FUNCTION_BLOCK FB_ProfidriveTelegram1_Test EXTENDS TcUnit.FB_TestSuite

Test_ProcessDataControl();
Test_ProcessDataStatus();

METHOD Test_ProcessDataControl : REFERENCE TO FB_Test
VAR
	fbDrive 					: FB_ProfidriveTelegram1;
	
	nExpectedSTW1 				: WORD;
	nExpectedNSOLL				: INT;
	nActualSTW1 				: WORD;
	nActualNSOLL				: INT;	
	
	aExpectedControlData 		: ARRAY[1..4] OF BYTE;
	aExpectedStatusData 		: ARRAY[1..4] OF BYTE;
END_VAR
TEST('Assign Process data Control');

//Arrange
nExpectedSTW1 := 16#A1B2;
nExpectedNSOLL 	:= UINT_TO_INT(16#C3D4);
F_Memcpy(ADR(aExpectedControlData), ADR(nExpectedSTW1), 2, FALSE);
F_Memcpy(ADR(aExpectedControlData) + 2, ADR(nExpectedNSOLL), 2, FALSE);
fbDrive.AssignProcessData(aExpectedControlData, aExpectedStatusData);

//Act
fbDrive.GetControlData();

//Assert
F_Memcpy(ADR(nActualSTW1), ADR(fbDrive.stControl), 2, FALSE);
F_Memcpy(ADR(nActualNSOLL), ADR(fbDrive.stControl) + 2, 2, FALSE);

AssertEquals(Expected := nExpectedSTW1,
             Actual := nActualSTW1,
             Message := 'nSTW1 is not correct');
	 
AssertEquals(Expected := nExpectedNSOLL,
             Actual := nActualNSOLL,
             Message := 'nNSOLL is not correct');	

TEST_FINISHED();


TEST('Assign Process data Control Swap');

//Arrange
nExpectedSTW1 := 16#C3F3;
nExpectedNSOLL 	:= UINT_TO_INT(16#C3F3);
F_Memcpy(ADR(aExpectedControlData), ADR(nExpectedSTW1), 2, TRUE);
F_Memcpy(ADR(aExpectedControlData) + 2, ADR(nExpectedNSOLL), 2, TRUE);

fbDrive.stConfig.bSwapProcessData := TRUE;
fbDrive.AssignProcessData(aExpectedControlData, aExpectedStatusData);

//Act
fbDrive.GetControlData();

//Assert
F_Memcpy(ADR(nActualSTW1), ADR(fbDrive.stControl), 2, FALSE);
F_Memcpy(ADR(nActualNSOLL), ADR(fbDrive.stControl) + 2, 2, FALSE);

AssertEquals(Expected := nExpectedSTW1,
             Actual := nActualSTW1,
             Message := 'nSTW1 is not correct');
	 
AssertEquals(Expected := nExpectedNSOLL,
             Actual := nActualNSOLL,
             Message := 'nNSOLL is not correct');	

TEST_FINISHED();
END_METHOD

METHOD Test_ProcessDataStatus : REFERENCE TO FB_Test
VAR
	fbDrive 					: FB_ProfidriveTelegram1;
	
	nExpectedZSW1 				: WORD;
	nExpectedNIST				: INT;	
	nActualZSW1 				: WORD;
	nActualNIST					: INT;	

	aExpectedControlData 		: ARRAY[1..4] OF BYTE;	
	aExpectedStatusData 		: ARRAY[1..4] OF BYTE;	
END_VAR
TEST('Assign Process data Status');

//Arrange
nExpectedZSW1 := 16#A1B2;
nExpectedNIST 	:= UINT_TO_INT(16#C3D4);
F_Memcpy(ADR(fbDrive.stStatus), ADR(nExpectedZSW1), 2, FALSE);
F_Memcpy(ADR(fbDrive.stStatus) + 2, ADR(nExpectedNIST), 2, FALSE);
fbDrive.AssignProcessData(aExpectedControlData, aExpectedStatusData);

//Act
fbDrive.SetStatusData();

//Assert
F_Memcpy(ADR(nActualZSW1), ADR(aExpectedStatusData), 2, FALSE);
F_Memcpy(ADR(nActualNIST), ADR(aExpectedStatusData) + 2, 2, FALSE);

AssertEquals(Expected := nExpectedZSW1,
             Actual := nActualZSW1,
             Message := 'nZSW1 is not correct');
	 
AssertEquals(Expected := nExpectedNIST,
             Actual := nActualNIST,
             Message := 'nNIST is not correct');	

TEST_FINISHED();


TEST('Assign Process data Status SWAP');

//Arrange
nExpectedZSW1 := 16#A1B2;
nExpectedNIST 	:= UINT_TO_INT(16#C3D4);
F_Memcpy(ADR(fbDrive.stStatus), ADR(nExpectedZSW1), 2, FALSE);
F_Memcpy(ADR(fbDrive.stStatus) + 2, ADR(nExpectedNIST), 2, FALSE);
fbDrive.AssignProcessData(aExpectedControlData, aExpectedStatusData);
fbDrive.stConfig.bSwapProcessData := TRUE;

//Act
fbDrive.SetStatusData();

//Assert
F_Memcpy(ADR(nActualZSW1), ADR(aExpectedStatusData), 2, TRUE);
F_Memcpy(ADR(nActualNIST), ADR(aExpectedStatusData) + 2, 2, TRUE);

AssertEquals(Expected := nExpectedZSW1,
             Actual := nActualZSW1,
             Message := 'nZSW1 is not correct');
	 
AssertEquals(Expected := nExpectedNIST,
             Actual := nActualNIST,
             Message := 'nNIST is not correct');	

TEST_FINISHED();
END_METHOD

END_FUNCTION_BLOCK

(* stored: Version 1.1.0.1, ProductVersion 3.1.4024.12
   POU FB_ProfidriveTelegram1_Test: Id {a3b4595a-ff1b-0df3-298e-dfe9bd1cbb12}, SpecialFunc None
   Method Test_ProcessDataControl: Id {16ebd94e-bdad-08df-3f30-2d8391d4539e}
   Method Test_ProcessDataStatus: Id {4abedd89-dcb3-0b8f-04ba-e93a9c2d32c9} *)
